(* IEC 61131-3 sources: Industry-PLC-LLM/data/PLCBEAD_repo/PLCBEAD_PLCEmbed-main/PLC-BEAD/Source/GEB/MULTIME, 1 file *)

(* ---- MULTIME.ST ---- *)
FUNCTION _REAL_TO_DWORD: DWORD

  VAR_INPUT
    X :	REAL;
  END_VAR

  IF REAL_TO_DWORD(0.5) = DWORD#1 THEN
    _REAL_TO_DWORD := REAL_TO_DWORD(X);
  ELSIF X > 0.0 THEN
    _REAL_TO_DWORD := REAL_TO_DWORD(X+0.5);
  ELSIF X < 0.0 THEN
    _REAL_TO_DWORD := REAL_TO_DWORD(X-0.5);
  ELSE
    _REAL_TO_DWORD := DWORD#0;
  END_IF;
END_FUNCTION

FUNCTION _DWORD_TO_REAL:REAL
	VAR_INPUT
		IN :	DWORD;
	END_VAR

	_DWORD_TO_REAL := UDINT_TO_REAL(DWORD_TO_UDINT(IN));

END_FUNCTION

FUNCTION MULTIME_B:TIME
	VAR_INPUT
		T :	TIME;
		M :	REAL;
	END_VAR

	MULTIME_B := DWORD_TO_TIME(_REAL_TO_DWORD(_DWORD_TO_REAL(TIME_TO_DWORD(T))*M));
END_FUNCTION

PROGRAM program0
  VAR
    LocalVar0 : TIME;
	LocalVaR1  : REAL;
	LocalOUT  : TIME;
  END_VAR
  	LocalOUT := MULTIME_B(LocalVar0, LocalVaR1 );
END_PROGRAM
